(* IEC 61131-3 sources: programs/VI-54/VI-54_20171205/VI-54_20171205/Stations/Screen/LseClass170718/Class/DiagnosticUserFunction_PLC, 1 file *)

(* ---- DiagnosticUserFunction_PLC.st ---- *)
(*!
<Class
	Name               = "DiagnosticUserFunction_PLC"
	Revision           = "1.0"
	RealtimeTask       = "false"
	CyclicTask         = "false"
	BackgroundTask     = "false"
	Sigmatek           = "false"
	OSInterface        = "false"
	HighPriority       = "false"
	Automatic          = "false"
	UpdateMode         = "Prescan"
	SharedCommandTable = "true"
	Objectsize         = "(540,120)"
	Comment            = "Use this class as base class for new functions of the diagnose.">
	<Channels>
		<Server Name="sStatus" Visualized="false" Initialize="false" WriteProtected="true" Retentive="false" Comment="Actual status."/>
	</Channels>
	<RevDoku>
		<Owner Company="Sigmatek"/>
		<Dokumentation Revision="1.0" Date="2016-06-02" Author="HötAnt" Company="Sigmatek" Description="Creation"/>
	</RevDoku>
</Class>
*)
DiagnosticUserFunction_PLC : CLASS
  //Servers:
	sStatus 	: SvrChCmd_iprStates;
  //Clients:
  //Variables:
  //Functions:
				//! <Function Comment="Is called when the diagnostic export starts." Name="StartWork"/>
	FUNCTION VIRTUAL GLOBAL StartWork
		VAR_OUTPUT
			retcode 	: iprStates;			//! <Variable Comment="Ready..Continue with the work methode&#13;&#10;Error..ssw is in a wrong step" Name="StartWork.retcode"/>
		END_VAR;
				//! <Function Comment="This method will be called cyclic when the diagnostic export is started." Name="WorkMethode"/>
	FUNCTION VIRTUAL GLOBAL WorkMethode;
				//! <Function Comment="Get the actual state of the function." Name="GetWorkState"/>
	FUNCTION VIRTUAL GLOBAL GetWorkState
		VAR_OUTPUT
			retcode 	: iprStates;			//! <Variable Comment="Actual state." Name="GetWorkState.retcode"/>
		END_VAR;
				//! <Function Comment="Method to get the actual error code." Name="GetErrorCode"/>
	FUNCTION VIRTUAL GLOBAL GetErrorCode
		VAR_OUTPUT
			retcode 	: _DiagErrorCode;			//! <Variable Comment="Error code." Name="GetErrorCode.retcode"/>
		END_VAR;
				//! <Function Comment="Method to get the size of the data which should be send." Name="GetDataSize"/>
	FUNCTION VIRTUAL GLOBAL GetDataSize
		VAR_OUTPUT
			retcode 	: UDINT;			//! <Variable Comment="Size of the data." Name="GetDataSize.retcode"/>
		END_VAR;
				//! <Function Comment="Method to get the pointer to the data of the user function." Name="GetDataPtr"/>
	FUNCTION VIRTUAL GLOBAL GetDataPtr
		VAR_OUTPUT
			dataPtr 	: ^void;			//! <Variable Comment="Pointer to the user data." Name="GetDataPtr.dataPtr"/>
		END_VAR;
				//! <Function Comment="Is called when the work method finished." Name="EndWork"/>
	FUNCTION VIRTUAL GLOBAL EndWork;
  //Tables:
	FUNCTION @STD
		VAR_OUTPUT
			ret_code	: CONFSTATES;
		END_VAR;
	FUNCTION GLOBAL TAB @CT_;
END_CLASS;

#pragma warning(disable:73);
#pragma warning(disable:76);

FUNCTION VIRTUAL GLOBAL DiagnosticUserFunction_PLC::WorkMethode

END_FUNCTION

FUNCTION VIRTUAL GLOBAL DiagnosticUserFunction_PLC::GetWorkState
	VAR_OUTPUT
		retcode 	: iprStates;
	END_VAR

END_FUNCTION

FUNCTION VIRTUAL GLOBAL DiagnosticUserFunction_PLC::GetErrorCode
	VAR_OUTPUT
		retcode 	: _DiagErrorCode;
	END_VAR

END_FUNCTION

FUNCTION VIRTUAL GLOBAL DiagnosticUserFunction_PLC::GetDataSize
	VAR_OUTPUT
		retcode 	: UDINT;
	END_VAR

END_FUNCTION

FUNCTION VIRTUAL GLOBAL DiagnosticUserFunction_PLC::GetDataPtr
	VAR_OUTPUT
		dataPtr 	: ^void;
	END_VAR

END_FUNCTION

FUNCTION VIRTUAL GLOBAL DiagnosticUserFunction_PLC::StartWork
	VAR_OUTPUT
		retcode 	: iprStates;
	END_VAR

END_FUNCTION

FUNCTION VIRTUAL GLOBAL DiagnosticUserFunction_PLC::EndWork

END_FUNCTION
#pragma warning(default:73);
#pragma warning(default:76);
